FUNCTION_BLOCK SimulationTwoPositionCylinderWithFeedback EXTENDS CyclicInstance IMPLEMENTS I_Cylinder
VAR
	Output_Extend AT %Q* : BOOL;
	Output_Retract AT %Q* : BOOL;
	Input_Extended AT %I* : BOOL;
	Input_Retracted AT %I* : BOOL;
	retract, extend : TON;
END_VAR

METHOD PUBLIC CyclicCall
VAR_INPUT
END_VAR
retract(IN:=Output_Retract,PT:=T#2S);
extend(IN:=Output_Extend,PT:=T#2S);

Input_Retracted := retract.Q;
Input_Extended := extend.Q;
END_METHOD

METHOD PUBLIC FullyExtend
VAR_INPUT
END_VAR
Output_Extend := TRUE;
Output_Retract := FALSE;
END_METHOD

METHOD PUBLIC FullyRetract
VAR_INPUT
END_VAR
Output_Extend := FALSE;
Output_Retract := TRUE;
END_METHOD

PROPERTY PUBLIC IsExtending : BOOL
GET
IsExtending := (Output_Extend and not IsFullyExtended);
END_GET
END_PROPERTY

PROPERTY PUBLIC IsFullyExtended : BOOL
GET
IsFullyExtended := extend.Q;
END_GET
END_PROPERTY

PROPERTY PUBLIC IsFullyRetracted : BOOL
GET
IsFullyRetracted := retract.Q;
END_GET
END_PROPERTY

PROPERTY PUBLIC IsRetracting : Bool
GET
IsRetracting := (Output_Retract and not IsFullyRetracted);
END_GET
END_PROPERTY

END_FUNCTION_BLOCK

(* stored: Version 1.1.0.1, ProductVersion 3.1.4024.12
   POU SimulationTwoPositionCylinderWithFeedback: Id {4ba2db27-fce4-4565-b565-d3a605b12851}, SpecialFunc None
   Method CyclicCall: Id {d4141caf-79e3-41a3-a051-24b88daad0ff}
   Method FullyExtend: Id {aabe8531-b126-436b-a038-6b4b271b6dff}
   Method FullyRetract: Id {0b2e47a9-a398-4830-aac1-657a6a90d481}
   Property IsExtending: Id {fe391868-040a-440c-9380-4c73bb813258}
   Get Get: Id {b9b5c861-720a-4ebc-aad4-048f577a4924}
   Property IsFullyExtended: Id {11851497-1dac-4364-b376-b12e023335ba}
   Get Get: Id {30cc687c-d123-45cb-bc41-7d222d4388af}
   Property IsFullyRetracted: Id {77627329-8854-478f-8fe1-1befb6fcbb0a}
   Get Get: Id {a7bc123d-a528-4d30-b08f-34d34ff7e129}
   Property IsRetracting: Id {c26d884b-1e73-4d6a-9a97-abbbca7faa7c}
   Get Get: Id {9adf0790-393a-41b0-858c-345ab5f15c51} *)
